// TIA Portal V19 export
FUNCTION_BLOCK "Door_FB"   // FB47, F_LAD
TITLE = Safety Door Handling
// v. 1.0
// stored: Access Published
   VAR_INPUT
      LS : Bool;   // Safety input of door
      EntryReq : Bool;   // Pb entry request
      EntryEnable : Bool;   // Entry enable (all device are in safestate)
      Reset : Bool;   // Door reset
      LockEnable : Bool;   // Input of EletricLock key inserted but not locked
      Existing : Bool := TRUE;   // Door exist
   END_VAR
   VAR_OUTPUT
      Unlock : Bool;   // Unlock output for EletricLock
   END_VAR
   VAR_IN_OUT
      Sts : "udt_DoorSts";
   END_VAR
   VAR
      xRE_Reset : Bool;
      Rearm : Bool;
      TON_Unlock : TON;
   END_VAR
   VAR_TEMP   // added for the SCL form of the ladder/FBD networks
      _w1 : Bool;
   END_VAR
BEGIN

REGION Network 1: Rearm Door (Normal Or LockDoor)
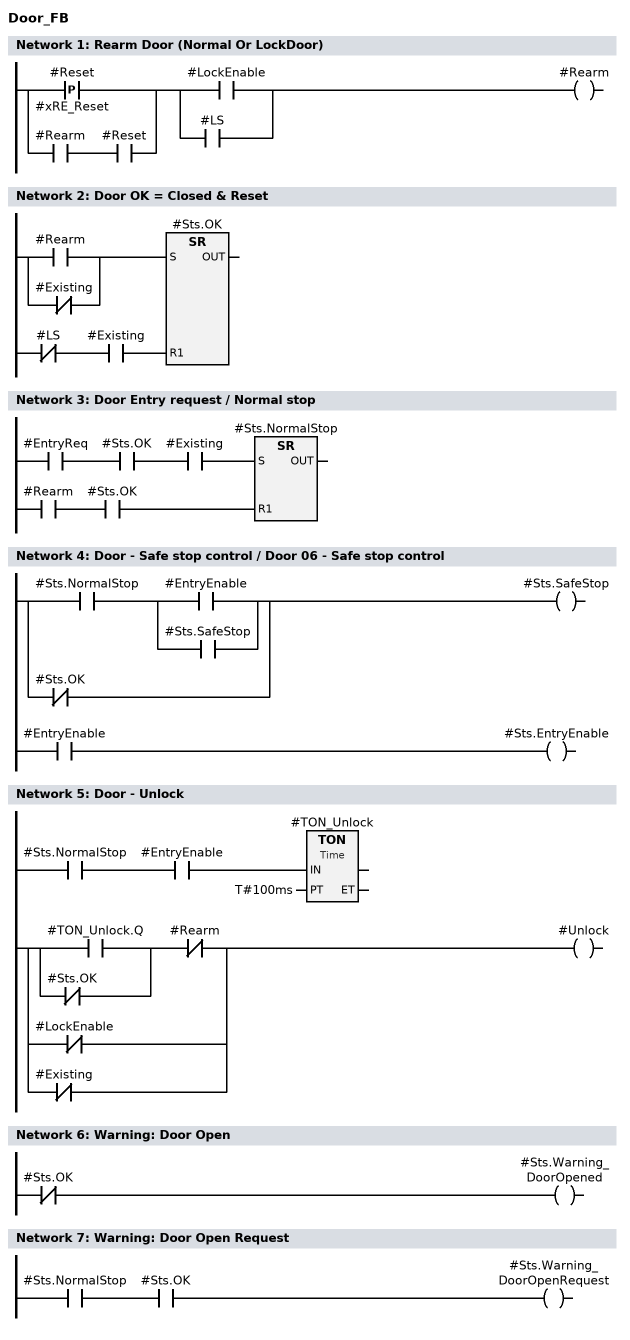
   RUNG wire#powerrail
      P_Contact(operand := #Reset, bit := #xRE_Reset)
      wire#w1
      Contact( #LockEnable )
      wire#w2
      Coil( #Rearm )
   END_RUNG
   RUNG wire#powerrail
      Contact( #Rearm )
      Contact( #Reset )
   END_RUNG wire#w1
   RUNG wire#w1
      Contact( #LS )
   END_RUNG wire#w2
   // the same network as SCL:
   #_w1 := #Reset AND NOT #xRE_Reset;   // rising edge of #Reset
   #xRE_Reset := #Reset;
   #Rearm := (#_w1 OR (#Rearm AND #Reset)) AND (#LockEnable OR #LS);
END_REGION

REGION Network 2: Door OK = Closed & Reset
   RUNG wire#powerrail
      Contact( #Rearm )
      wire#w1
      S_SR(operand := #Sts.OK, r1 := wire#w2)
   END_RUNG
   RUNG wire#powerrail
      I_Contact( #Existing )
   END_RUNG wire#w1
   RUNG wire#powerrail
      I_Contact( #LS )
      Contact( #Existing )
   END_RUNG wire#w2
   // the same network as SCL:
   IF #Rearm OR NOT #Existing THEN
       #Sts.OK := TRUE;   // SR flip-flop
   END_IF;
   IF NOT #LS AND #Existing THEN #Sts.OK := FALSE; END_IF;
END_REGION

REGION Network 3: Door Entry request / Normal stop
   RUNG wire#powerrail
      Contact( #EntryReq )
      Contact( #Sts.OK )
      Contact( #Existing )
      S_SR(operand := #Sts.NormalStop, r1 := wire#w1)
   END_RUNG
   RUNG wire#powerrail
      Contact( #Rearm )
      Contact( #Sts.OK )
   END_RUNG wire#w1
   // the same network as SCL:
   IF #EntryReq AND #Sts.OK AND #Existing THEN
       #Sts.NormalStop := TRUE;   // SR flip-flop
   END_IF;
   IF #Rearm AND #Sts.OK THEN #Sts.NormalStop := FALSE; END_IF;
END_REGION

REGION Network 4: Door - Safe stop control / Door 06 - Safe stop control
   RUNG wire#powerrail
      Contact( #Sts.NormalStop )
      wire#w1
      Contact( #EntryEnable )
      wire#w2
      Coil( #Sts.SafeStop )
   END_RUNG
   RUNG wire#w1
      Contact( #Sts.SafeStop )
   END_RUNG wire#w2
   RUNG wire#powerrail
      I_Contact( #Sts.OK )
   END_RUNG wire#w2
   RUNG wire#powerrail
      Contact( #EntryEnable )
      Coil( #Sts.EntryEnable )
   END_RUNG
   // the same network as SCL:
   #Sts.SafeStop := (#Sts.NormalStop AND (#EntryEnable OR #Sts.SafeStop)) OR NOT #Sts.OK;
   #Sts.EntryEnable := #EntryEnable;
END_REGION

REGION Network 5: Door - Unlock
   RUNG wire#powerrail
      Contact( #Sts.NormalStop )
      Contact( #EntryEnable )
      { S7_Templates := "[time_type := Time, codedbool_type := DInt]" } #TON_Unlock.TON(pt := T#100ms, et =>)
   END_RUNG
   RUNG wire#powerrail
      Contact( #TON_Unlock.Q )
      wire#w1
      I_Contact( #Rearm )
      wire#w2
      Coil( #Unlock )
   END_RUNG
   RUNG wire#powerrail
      I_Contact( #Sts.OK )
   END_RUNG wire#w1
   RUNG wire#powerrail
      I_Contact( #LockEnable )
   END_RUNG wire#w2
   RUNG wire#powerrail
      I_Contact( #Existing )
   END_RUNG wire#w2
   // the same network as SCL:
   #TON_Unlock.TON(IN := #Sts.NormalStop AND #EntryEnable, PT := T#100ms);
   #Unlock := ((#TON_Unlock.Q OR NOT #Sts.OK) AND NOT #Rearm) OR NOT #LockEnable OR NOT #Existing;
END_REGION

REGION Network 6: Warning: Door Open
   RUNG wire#powerrail
      I_Contact( #Sts.OK )
      Coil( #Sts.Warning_DoorOpened )
   END_RUNG
   // the same network as SCL:
   #Sts.Warning_DoorOpened := NOT #Sts.OK;
END_REGION

REGION Network 7: Warning: Door Open Request
   RUNG wire#powerrail
      Contact( #Sts.NormalStop )
      Contact( #Sts.OK )
      Coil( #Sts.Warning_DoorOpenRequest )
   END_RUNG
   // the same network as SCL:
   #Sts.Warning_DoorOpenRequest := #Sts.NormalStop AND #Sts.OK;
END_REGION
END_FUNCTION_BLOCK
